(* Logix 5000 project; controller PLC2_Project2_2 Emulate 5570 rev 20.11; software revision 20.00 *)
// Same project, using tutor's method for the program.

TASK MainTask (continuous, watchdog 500 ms) : MainProgram

MODULES
   Local : Emulate 5570 (ICP 1, rev 20.11)
      Simulator_Card : vendor 1 type 0 code 15 (ICP 2, rev 1.1, Output RPI 5 ms)
END_MODULES

PROGRAM MainProgram   (* main routine MainRoutine *)
VAR
   Cycle_Stage : DINT;   // Cycle Stage: 0 = Bring Box 1 = Fill Box 2 = Unload Station 3 = Intermediate
   FillBox_ONS : BOOL;
   Motor_En : BOOL;
   Motor_Interrupt : BOOL;
   Motor_ONS : BOOL;
   Motor_StartTrigger : BOOL;
   MoveBox_ONS : BOOL;
   Pecan_ONS : BOOL;
   PecanHopper_En : BOOL;
   PecanHopper_OpenTrigger : BOOL;
   Switch_BluePhotoEye : BOOL;
   Switch_Level : BOOL;
   Switch_Proximity : BOOL;
   Switch_RedPhotoEye : BOOL;
   Walnut_ONS : BOOL;
   WalnutHopper_En : BOOL;
   WalnutHopper_OpenTrigger : BOOL;
END_VAR

ROUTINE Controls   (* ladder *)
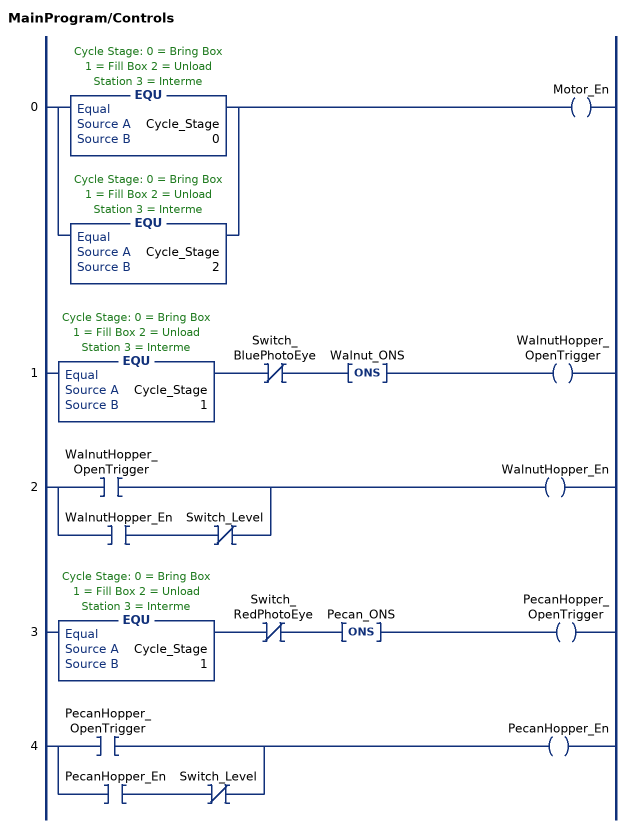
   0: [EQU(Cycle_Stage,0) ,EQU(Cycle_Stage,2) ]OTE(Motor_En);
   1: EQU(Cycle_Stage,1)XIO(Switch_BluePhotoEye)ONS(Walnut_ONS)OTE(WalnutHopper_OpenTrigger);
   2: [XIC(WalnutHopper_OpenTrigger) ,XIC(WalnutHopper_En) XIO(Switch_Level) ]OTE(WalnutHopper_En);
   3: EQU(Cycle_Stage,1)XIO(Switch_RedPhotoEye)ONS(Pecan_ONS)OTE(PecanHopper_OpenTrigger);
   4: [XIC(PecanHopper_OpenTrigger) ,XIC(PecanHopper_En) XIO(Switch_Level) ]OTE(PecanHopper_En);
END_ROUTINE

ROUTINE Cycle   (* ladder *)
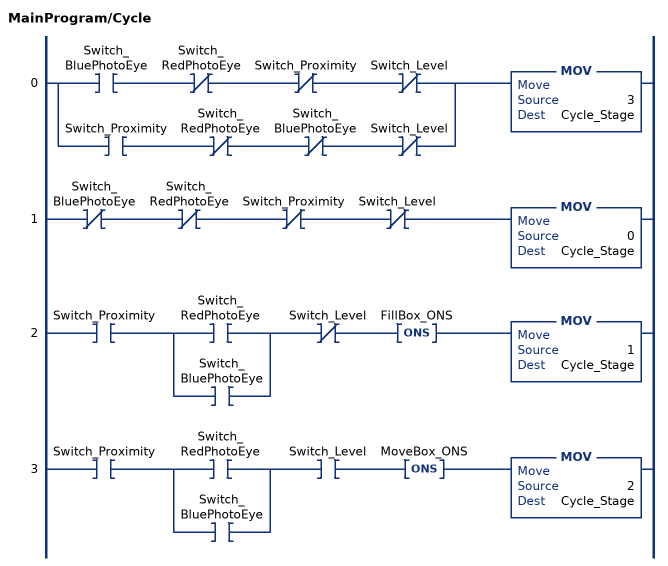
   0: [XIC(Switch_BluePhotoEye) XIO(Switch_RedPhotoEye) XIO(Switch_Proximity) XIO(Switch_Level) ,XIC(Switch_Proximity) XIO(Switch_RedPhotoEye) XIO(Switch_BluePhotoEye) XIO(Switch_Level) ]MOV(3,Cycle_Stage);
   1: XIO(Switch_BluePhotoEye)XIO(Switch_RedPhotoEye)XIO(Switch_Proximity)XIO(Switch_Level)MOV(0,Cycle_Stage);
   2: XIC(Switch_Proximity)[XIC(Switch_RedPhotoEye) ,XIC(Switch_BluePhotoEye) ]XIO(Switch_Level)ONS(FillBox_ONS)MOV(1,Cycle_Stage);
   3: XIC(Switch_Proximity)[XIC(Switch_RedPhotoEye) ,XIC(Switch_BluePhotoEye) ]XIC(Switch_Level)ONS(MoveBox_ONS)MOV(2,Cycle_Stage);
END_ROUTINE

ROUTINE InputOutput   (* ladder *)
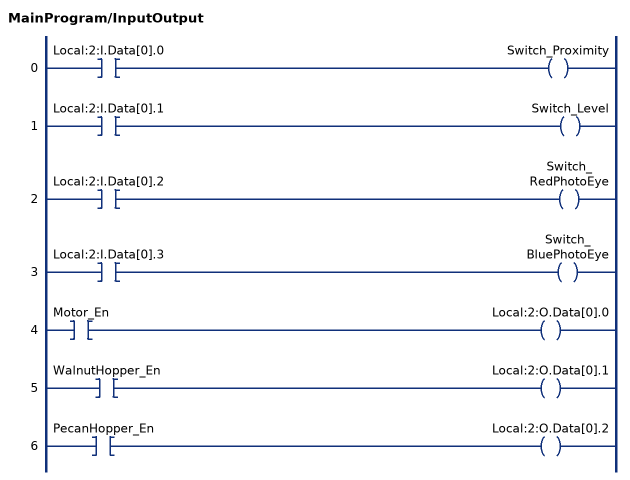
   0: XIC(Local:2:I.Data[0].0)OTE(Switch_Proximity);
   1: XIC(Local:2:I.Data[0].1)OTE(Switch_Level);
   2: XIC(Local:2:I.Data[0].2)OTE(Switch_RedPhotoEye);
   3: XIC(Local:2:I.Data[0].3)OTE(Switch_BluePhotoEye);
   4: XIC(Motor_En)OTE(Local:2:O.Data[0].0);
   5: XIC(WalnutHopper_En)OTE(Local:2:O.Data[0].1);
   6: XIC(PecanHopper_En)OTE(Local:2:O.Data[0].2);
END_ROUTINE

ROUTINE MainRoutine   (* ladder *)
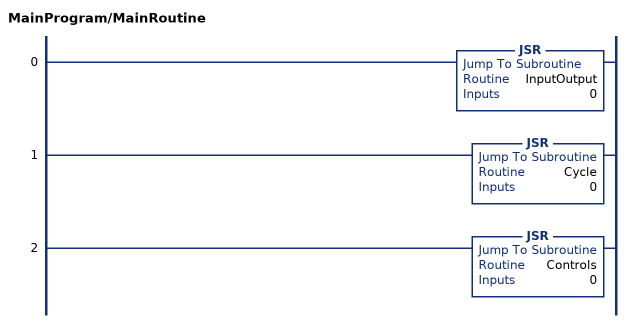
   0: JSR(InputOutput,0);
   1: JSR(Cycle,0);
   2: JSR(Controls,0);
END_ROUTINE
END_PROGRAM
